FUNCTION_BLOCK BaseComponent
VAR_INPUT
END_VAR
VAR_OUTPUT
END_VAR
VAR
END_VAR

END_FUNCTION_BLOCK

(* stored: Version 1.1.0.1
   POU BaseComponent: Id {5e455814-cab3-4c57-bf18-d03963995e63}, SpecialFunc None *)
